(* CODESYS project IFTTT Test Lib 1.1.ecp

Project tree, tasks and I/O mapping:
  Controller : 750-8212 PFC200 2ETH RS, WAGO, order no. 0750-8212, version 5.13.2.22
    application Application
      libraries: ; IFTTT_Lib, 1.1 (Kurt Braun)
      task PLC_Task (cyclic, interval t#50ms, priority 15) calls PLC_PRG
      program PLC_PRG [ST]
    Kbus : Kbus, WAGO, version 1.4.0.2
        unmapped channels: K-BUS diagnostics
      _8_DO_DI_Generic : 075x-8DO8DI, WAGO, order no. 075x-8DO8DI, version 0.0.0.13
          settings: K-BUS Module slot index = 1
          input  xDI1 : BOOL  // _IN._IN
          unmapped channels: _IN, _OUT
    MODBUS
      MODBUS : MODBUS, WAGO, order no. n/a, version 1.1.1.15
    Common.PCI
    Serial
      COM1 : COM1, WAGO, version 0.0.0.19
*)

// Controller/Application/PLC_PRG
PROGRAM PLC_PRG
VAR
	sValue1 : STRING := 'Hello ';
	sValue2 : STRING := 'World ';
	sValue3 : STRING := '!';
	sKey : STRING := 'dScfmjG8sTQuYYjcgHrCCw';
	sEvent : STRING := 'email';
	xError : BOOL;
	xSent : BOOL;
	sStatus : STRING;
	IFTTT_Send_Email : IFTTT_Lib.IFTTT_Send;
END_VAR

IFTTT_Send_Email(
	sValue1 := sValue1,
	sValue2 := sValue2,
	sValue3 := sValue3,
	sEvent := sEvent,
	sKey := sKey,
	xSend := xDI1,
	xError => xError,
	xSent => xSent,
	sReturn_String => sStatus);

END_PROGRAM
